// TIA Portal project "systemVariables" (V19)

(* hardware
DEVICE "HMI_1"  TP700 Comfort
   slot 0: "HMI_1"  TP700 Comfort  6AV2 124-0GC01-0AX0  17.0.0.0
   slot 1: "HMI_RT_1"  TP700 Comfort  6AV2 124-0GC01-0AX0  17.0.0.0
   slot 5: "HMI_1.IE_CP_1"  PROFINET Interface  17.0.0.0
      slot 1: "PROFINET Interface_1"  PROFINET Interface
         slot 1: "Port_1"  Port
         slot 2: "Port_2"  Port
   slot 7: "HMI_1.MPI/DP_CP_1"  MPI/DP Interface  17.0.0.0
DEVICE "S7-1500/ET200MP station_1"  S7-1500 station
   slot 0: "Rail_0"  Rack  6ES7 590-1***0-0AA0
   slot 1: "PLC_1"  CPU 1511-1 PN  6ES7 511-1AK00-0AB0  V1.8
      slot 3: "CPU display_1"  6ES7591-1AA00-0AA0
      slot 32768: "PROFINET interface_1"  X1
         slot 32769: "Port_1"  X1 P1
         slot 32770: "Port_2"  X1 P2
*)

// ===== PLC "PLC_1"  CPU 1511-1 PN =====

VAR_GLOBAL   // PLC tag table "Default tag table"
   "alwayOff" AT %M0.0 : Bool;   // Always Off
   "alwaysOn" AT %M0.1 : Bool;   // Always On
   "firstScan" AT %M0.2 : Bool;   // First Scan
   "afterFirstScan" AT %M0.4 : Bool;   // After First Scan
   "clock1Hz" AT %M0.6 : Bool;   // Clock 60Hz
   "clockHour" AT %MW20 : UInt;   // Clock Hour
   "clockMinute" AT %MW22 : UInt;   // Clock Minutes
   "clockSecond" AT %MW24 : UInt;   // Clock Seconds
   "clockDay" AT %MW26 : UInt;
   "clockMonth" AT %MW28 : UInt;
   "clockYear" AT %MW30 : UInt;
   "test" AT %MD2 : Real;
END_VAR

DATA_BLOCK "systemVariables_DB"   // DB1
{ S7_Optimized_Access := 'TRUE' }
VERSION : 0.1
   VAR
      "timer" : Array[0..31] of IEC_TIMER;
      pulse : Array[0..31] of Bool;
      actualTime : DTL;
   END_VAR
BEGIN
END_DATA_BLOCK

DATA_BLOCK "Clock_DB"   // DB2
{ S7_Optimized_Access := 'TRUE' }
VERSION : 0.1
// stored: InstanceOfName Clock
"Clock"
BEGIN
END_DATA_BLOCK

FUNCTION_BLOCK "Clock"   // FB1, SCL
{ S7_Optimized_Access := 'TRUE' }
VERSION : 0.1
   VAR_OUTPUT
      bissexto : Bool;
      dayOfMonth : Int;
   END_VAR
   VAR_IN_OUT
      hours : UInt;
      minutes : UInt;
      seconds : UInt;
      day : UInt;
      month : UInt;
      year : UInt;
      dtl : DTL;
   END_VAR
   VAR
      tAtual : Time := T#0s;
      tIncremento : Time := T#1s;
      temporizador : TON_TIME;
      auxBissexto1 : Int;
      auxBissexto2 : Int;
      auxBissexto3 : Int;
   END_VAR
   VAR_TEMP
      lastsecond : Int;   // Last Second
      fev : Int;
   END_VAR
BEGIN
   // Calculo ano bissexto
   #auxBissexto1 := #year / 4;
   #auxBissexto2 := #year / 100;
   #auxBissexto3 := #year / 400;

   IF (#auxBissexto1 * 4) = #year AND (#auxBissexto2 * 100) < #year THEN

       #bissexto := 1;

   END_IF;

   IF (#auxBissexto1 * 4) = #year AND (#auxBissexto2 * 100) = #year AND (#auxBissexto3 * 400) = #year THEN

       #bissexto := 1;

   END_IF;

   IF #bissexto = 1 AND #month = 2 THEN

       #dayOfMonth := 29;

   ELSE

       #dayOfMonth := 28;
       #bissexto := 0;

   END_IF;

   CASE #month OF
       1, 3, 5, 7, 8, 10, 12:
           #dayOfMonth := 31;

       4, 6, 9, 11:
           #dayOfMonth := 30;

   END_CASE;

   // Clock
   // 
   #temporizador(IN := TRUE, PT := T#1s);

   IF #temporizador.Q THEN
       #temporizador(IN := FALSE,
                     PT := t#1s);

       #seconds := #seconds + 1;

       IF #seconds >= 60 THEN
           #seconds := 0;
           #minutes := #minutes + 1;

           IF #minutes >= 60 THEN
               #minutes := 0;
               #hours := #hours + 1;

               IF #hours >= 24 THEN
                   #hours := 0;
                   #day := #day + 1;

                   IF #day >= #dayOfMonth THEN
                       #day := 1;
                       #month := #month + 1;

                       IF #month >= 12 THEN
                           #month := 1;
                           #year := #year + 1;

                       END_IF;
                   END_IF;
               END_IF;
           END_IF;
       END_IF;
   END_IF;

   //DTL write
   //
   #dtl.SECOND := #seconds;
   #dtl.MINUTE := #minutes;
   #dtl.HOUR := #hours;

   #dtl.DAY := #day;
   #dtl.MONTH := #month;
   #dtl.YEAR := #year;
END_FUNCTION_BLOCK

FUNCTION "systemVariables" : Void   // FC1, LAD
{ S7_Optimized_Access := 'TRUE' }
VERSION : 0.1
   VAR CONSTANT
      timers : LTime;   // timers
   END_VAR
   VAR_TEMP   // added for the SCL form of the ladder/FBD networks
      _w1 : Bool;
   END_VAR
BEGIN

REGION Network 1: Always Off
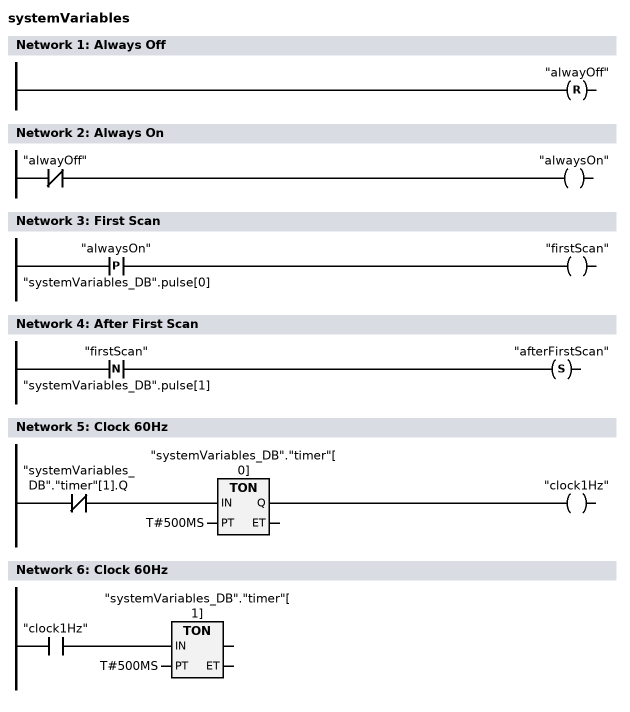
   RUNG wire#powerrail
      R_Coil( "alwayOff" )
   END_RUNG
   // the same network as SCL:
   "alwayOff" := FALSE;
END_REGION

REGION Network 2: Always On
   RUNG wire#powerrail
      I_Contact( "alwayOff" )
      Coil( "alwaysOn" )
   END_RUNG
   // the same network as SCL:
   "alwaysOn" := NOT "alwayOff";
END_REGION

REGION Network 3: First Scan
   RUNG wire#powerrail
      P_Contact(operand := "alwaysOn", bit := "systemVariables_DB".pulse[0])
      Coil( "firstScan" )
   END_RUNG
   // the same network as SCL:
   #_w1 := "alwaysOn" AND NOT "systemVariables_DB".pulse[0];   // rising edge of "alwaysOn"
   "systemVariables_DB".pulse[0] := "alwaysOn";
   "firstScan" := #_w1;
END_REGION

REGION Network 4: After First Scan
   RUNG wire#powerrail
      N_Contact(operand := "firstScan", bit := "systemVariables_DB".pulse[1])
      S_Coil( "afterFirstScan" )
   END_RUNG
   // the same network as SCL:
   #_w1 := NOT "firstScan" AND "systemVariables_DB".pulse[1];   // falling edge of "firstScan"
   "systemVariables_DB".pulse[1] := "firstScan";
   IF #_w1 THEN "afterFirstScan" := TRUE; END_IF;
END_REGION

REGION Network 5: Clock 60Hz
   "systemVariables_DB"."timer"[0].TON(IN := NOT "systemVariables_DB"."timer"[1].Q, PT := T#500MS);
   "clock1Hz" := "systemVariables_DB"."timer"[0].Q;
END_REGION

REGION Network 6: Clock 60Hz
   "systemVariables_DB"."timer"[1].TON(IN := "clock1Hz", PT := T#500MS);
END_REGION
END_FUNCTION

ORGANIZATION_BLOCK "Main"   // OB1, LAD, ProgramCycle
TITLE = "Main Program Sweep (Cycle)"
{ S7_Optimized_Access := 'TRUE' }
VERSION : 0.1
   VAR_INPUT
      Initial_Call : Bool;   // Initial call of this OB
      Remanence : Bool;   // =True, if remanent data are available
   END_VAR
BEGIN

REGION Network 1
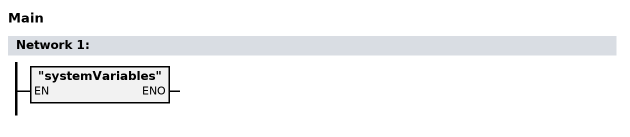
   RUNG wire#powerrail
      "systemVariables"()
   END_RUNG
   // the same network as SCL:
   "systemVariables"();
END_REGION

REGION Network 2 (SCL): Watch
   "Clock_DB"(hours:= "clockHour",
              minutes:= "clockMinute",
              seconds:= "clockSecond",
              day:= "clockDay",
              month:= "clockMonth",
              year:= "clockYear",
              "dtl":= "systemVariables_DB".actualTime );
END_REGION
END_ORGANIZATION_BLOCK

(* ===== HMI "HMI_RT_1" =====
system functions are stored by id; their names below are inferred from use

HMI tags "Default tag table"
   "Tag_ScreenNumber" : UInt, internal
   "clockHour" : UInt = PLC clockHour AT %MW20

screen "Root screen" 800x420, template "Template_1"
   on GenerateScreen: SetTag("Tag_ScreenNumber", 1)
   TextField "HmiScreenItemData_1" at 80,166 size 640x25; Text 'Welcome to HMI_1 (TP700 Comfort)!'
   Button "HmiScreenItemData" at 36,36 size 159x47; TextOff 'Screen0'; PictureOff "Navigates to Screen0 for TP700 Comfort 17.0.0.0"; PictureOn "Navigates to Screen0 for TP700 Comfort 17.0.0.0"
      on Release: ActivateScreen("Screen0", 0)
   Button "HmiScreenItemData_2" at 36,95 size 159x47; TextOff 'System screens'; PictureOff "Navigates to System screens for TP700 Comfort 17.0.0.0"; PictureOn "Navigates to System screens for TP700 Comfort 17.0.0.0"
      on Release: ActivateScreen("System screens", 0)

Template "Template_1" 800x420
   Button "Exit" at 720,360 size 78x58; TextOff 'Exit'; PictureOff "ExitRuntime_TP700_Comfort_TR"; PictureOn "ExitRuntime_TP700_Comfort_TR"
      on Release: StopRuntime(0)
   Button "Template_Button" at 640,360 size 78x58; TextOff 'Text'
   Button "Template_Button_1" at 560,360 size 78x58; TextOff 'Text'
   Button "Template_Button_2" at 480,360 size 78x58; TextOff 'Text'
   Button "Template_Button_3" at 400,360 size 78x58; TextOff 'Text'
   Button "Template_Button_4" at 321,360 size 78x58; TextOff 'Text'
   Button "Template_Button_5" at 241,360 size 78x58; TextOff 'Text'
   Button "Template_Button_6" at 161,360 size 78x58; TextOff 'Text'
   Button "Alarms" at 81,360 size 78x58; TextOff 'Alarms'; PictureOff "AlarmDisplay_TP700_Comfort_TR"; PictureOn "AlarmDisplay_TP700_Comfort_TR"
      on Release: function_ef3f5d25("Alarm window_Unacknowledged", -1)
   Button "Start screen" at 1,360 size 78x58; TextOff 'Start screen'; PictureOff "NavigateHome_TP700_Comfort_TR"; PictureOn "NavigateHome_TP700_Comfort_TR"
      on Release: ActivateScreen("Root screen", 0)

screen "Screen0" 800x420, template "Template_1"
   on GenerateScreen: SetTag("Tag_ScreenNumber", 2)
   Button "Back" at 1,1 size 159x47; TextOff 'Back'
      on Release: ActivateScreen("Root screen", 0)
   Button "HmiScreenItemData_1" at 36,95 size 159x47; TextOff 'Screen1'; PictureOff "Navigates to Screen1 for TP700 Comfort 17.0.0.0"; PictureOn "Navigates to Screen1 for TP700 Comfort 17.0.0.0"
      on Release: ActivateScreen("Screen1", 0)
   TextField "Text field_1" at 255,61 size 94x23; Text 'PLC Clock'
   IOField "I/O field_1" at 260,84 size 96x32; FormatPattern 99999
      ProcessValue <- "clockHour"

screen "Screen1" 800x420, template "Template_1"
   on GenerateScreen: SetTag("Tag_ScreenNumber", 3)
   TextField "HmiScreenItemData" at 80,166 size 640x25; Text 'Screen1'
   Button "Back" at 1,1 size 159x47; TextOff 'Back'
      on Release: ActivateScreen("Screen0", 0)

screen "System screens" 800x420, template "Template_1"
   on GenerateScreen: SetTag("Tag_ScreenNumber", 4)
   Button "Back" at 1,1 size 159x47; TextOff 'Back'
      on Release: ActivateScreen("Root screen", 0)
   Button "HmiScreenItemData" at 36,95 size 159x47; TextOff 'SIMATIC PLC system diagnos...'; PictureOff "Navigates to SIMATIC PLC system diagnostics for TP700 Comfort 17.0.0.0"; PictureOn "Navigates to SIMATIC PLC system diagnostics for TP700 Comfort 17.0.0.0"
      on Release: ActivateScreen("SIMATIC PLC system diagnostics", 0)
   Button "HmiScreenItemData_1" at 36,154 size 159x47; TextOff 'Project information'; PictureOff "Navigates to Project information for TP700 Comfort 17.0.0.0"; PictureOn "Navigates to Project information for TP700 Comfort 17.0.0.0"
      on Release: ActivateScreen("Project information", 0)
   Button "HmiScreenItemData_2" at 36,213 size 159x47; TextOff 'System settings'; PictureOff "Navigates to System settings for TP700 Comfort 17.0.0.0"; PictureOn "Navigates to System settings for TP700 Comfort 17.0.0.0"
      on Release: ActivateScreen("System settings", 0)
   Button "HmiScreenItemData_3" at 36,272 size 159x47; TextOff 'System information'; PictureOff "Navigates to System information for TP700 Comfort 17.0.0.0"; PictureOn "Navigates to System information for TP700 Comfort 17.0.0.0"
      on Release: ActivateScreen("System information", 0)

screen "SIMATIC PLC system diagnostics" 800x420, template "Template_1"
   on GenerateScreen: SetTag("Tag_ScreenNumber", 5)
   SysDiagControl "HmiScreenItemData" at 1,49 size 796x304
   Button "Back" at 1,1 size 159x47; TextOff 'Back'
      on Release: ActivateScreen("System screens", 0)

screen "Project information" 800x420, template "Template_1"
   on GenerateScreen: SetTag("Tag_ScreenNumber", 6)
   TextField "HmiScreenItemData" at 35,51 size 171x28; Text 'Project name:'
   TextField "HmiScreenItemData_1" at 241,51 size 524x28; Text 'systemVariables'
   TextField "HmiScreenItemData_2" at 35,81 size 171x28; Text 'Created on:'
   TextField "HmiScreenItemData_3" at 241,81 size 524x28; Text '6/10/2025 9:14:13 AM'
   TextField "HmiScreenItemData_4" at 35,111 size 171x28; Text 'Author:'
   TextField "HmiScreenItemData_5" at 241,111 size 524x28; Text 'Administrador'
   TextField "HmiScreenItemData_6" at 35,141 size 171x28; Text 'Description:'
   TextField "HmiScreenItemData_7" at 241,141 size 524x28; Text '(not configured)'
   Button "Back" at 1,1 size 159x47; TextOff 'Back'
      on Release: ActivateScreen("System screens", 0)

screen "System settings" 800x420, template "Template_1"
   on GenerateScreen: SetTag("Tag_ScreenNumber", 7)
   Button "Calibrate screen" at 36,95 size 159x47; TextOff 'Calibrate screen'
      on Release: function_bc3e350c()
   Button "Clean screen" at 36,154 size 159x47; TextOff 'Clean screen'
      on Release: function_be740847(30)
   Button "Back" at 1,1 size 159x47; TextOff 'Back'
      on Release: ActivateScreen("System screens", 0)

screen "System information" 800x420, template "Template_1"
   on GenerateScreen: SetTag("Tag_ScreenNumber", 8)
   TextField "HmiScreenItemData" at 35,51 size 171x28; Text 'HMI device type:'
   TextField "HmiScreenItemData_1" at 241,51 size 524x28; Text 'TP700 Comfort 17.0.0.0'
   TextField "HmiScreenItemData_2" at 35,81 size 171x28; Text 'Version:'
   TextField "HmiScreenItemData_3" at 35,111 size 171x28; Text 'Connection:'
   TextField "HmiScreenItemData_4" at 241,111 size 524x28; Text 'ETHERNET'
   TextField "HmiScreenItemData_5" at 35,141 size 171x28; Text 'PLC:'
   TextField "HmiScreenItemData_6" at 241,141 size 524x28; Text 'SIMATIC S7 1200'
   Button "Display version" at 241,81 size 524x28; TextOff 'Display version'
      on Release: function_febcb963(-1)
   Button "Back" at 1,1 size 159x47; TextOff 'Back'
      on Release: ActivateScreen("System screens", 0)
*)